// TIA Portal V20 export
FUNCTION_BLOCK "Simulation"   // FB191, LAD
// stored: MemoryReserve 100, Namespace Unit1.Em3, SetENOAutomatically false
   VAR_INPUT
      simulation { ExternalAccessible := 'False'; ExternalVisible := 'False'; ExternalWritable := 'False'} : Bool;
   END_VAR
   VAR
      instActuator { ExternalAccessible := 'False'; ExternalVisible := 'False'; ExternalWritable := 'False'} : Array[0..19] of "Simulation_Actuator";
      statDigitalSignal { ExternalAccessible := 'False'; ExternalVisible := 'False'; ExternalWritable := 'False'} : Array[0..9] of Bool;
   END_VAR
   VAR_TEMP
      tempJRPnPRightplace : Bool;
   END_VAR
   VAR_TEMP   // added for the SCL form of the ladder/FBD networks
      _w1 : Bool;
   END_VAR
BEGIN

REGION Network 1: Digital Signal
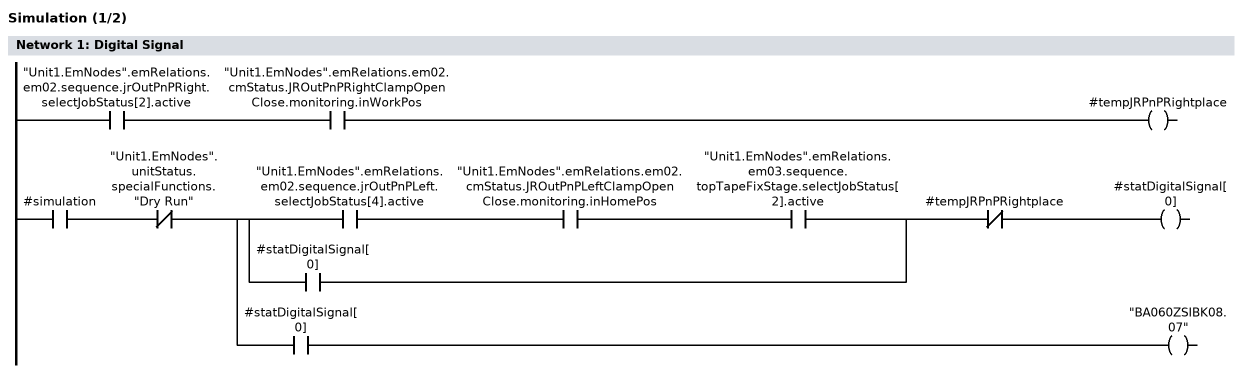
   RUNG wire#powerrail
      Contact( "Unit1.EmNodes".emRelations.em02.sequence.jrOutPnPRight.selectJobStatus[2].active )
      Contact( "Unit1.EmNodes".emRelations.em02.cmStatus.JROutPnPRightClampOpenClose.monitoring.inWorkPos )
      Coil( #tempJRPnPRightplace )
   END_RUNG
   RUNG wire#powerrail
      Contact( #simulation )
      I_Contact( "Unit1.EmNodes".unitStatus.specialFunctions."Dry Run" )
      wire#w1
      Contact( "Unit1.EmNodes".emRelations.em02.sequence.jrOutPnPLeft.selectJobStatus[4].active )
      Contact( "Unit1.EmNodes".emRelations.em02.cmStatus.JROutPnPLeftClampOpenClose.monitoring.inHomePos )
      Contact( "Unit1.EmNodes".emRelations.em03.sequence.topTapeFixStage.selectJobStatus[2].active )
      wire#w2
      I_Contact( #tempJRPnPRightplace )
      Coil( #statDigitalSignal[0] )
   END_RUNG
   RUNG wire#w1
      Contact( #statDigitalSignal[0] )
   END_RUNG wire#w2
   RUNG wire#w1
      Contact( #statDigitalSignal[0] )
      Coil( "BA060ZSIBK08.07" )
   END_RUNG
   // the same network as SCL:
   #tempJRPnPRightplace := "Unit1.EmNodes".emRelations.em02.sequence.jrOutPnPRight.selectJobStatus[2].active AND "Unit1.EmNodes".emRelations.em02.cmStatus.JROutPnPRightClampOpenClose.monitoring.inWorkPos;
   #_w1 := #simulation AND NOT "Unit1.EmNodes".unitStatus.specialFunctions."Dry Run";
   #statDigitalSignal[0] := #_w1 AND (("Unit1.EmNodes".emRelations.em02.sequence.jrOutPnPLeft.selectJobStatus[4].active AND "Unit1.EmNodes".emRelations.em02.cmStatus.JROutPnPLeftClampOpenClose.monitoring.inHomePos AND "Unit1.EmNodes".emRelations.em03.sequence.topTapeFixStage.selectJobStatus[2].active) OR #statDigitalSignal[0]) AND NOT #tempJRPnPRightplace;
   "BA060ZSIBK08.07" := #_w1 AND #statDigitalSignal[0];
END_REGION

REGION Network 2: Two Way Actuator
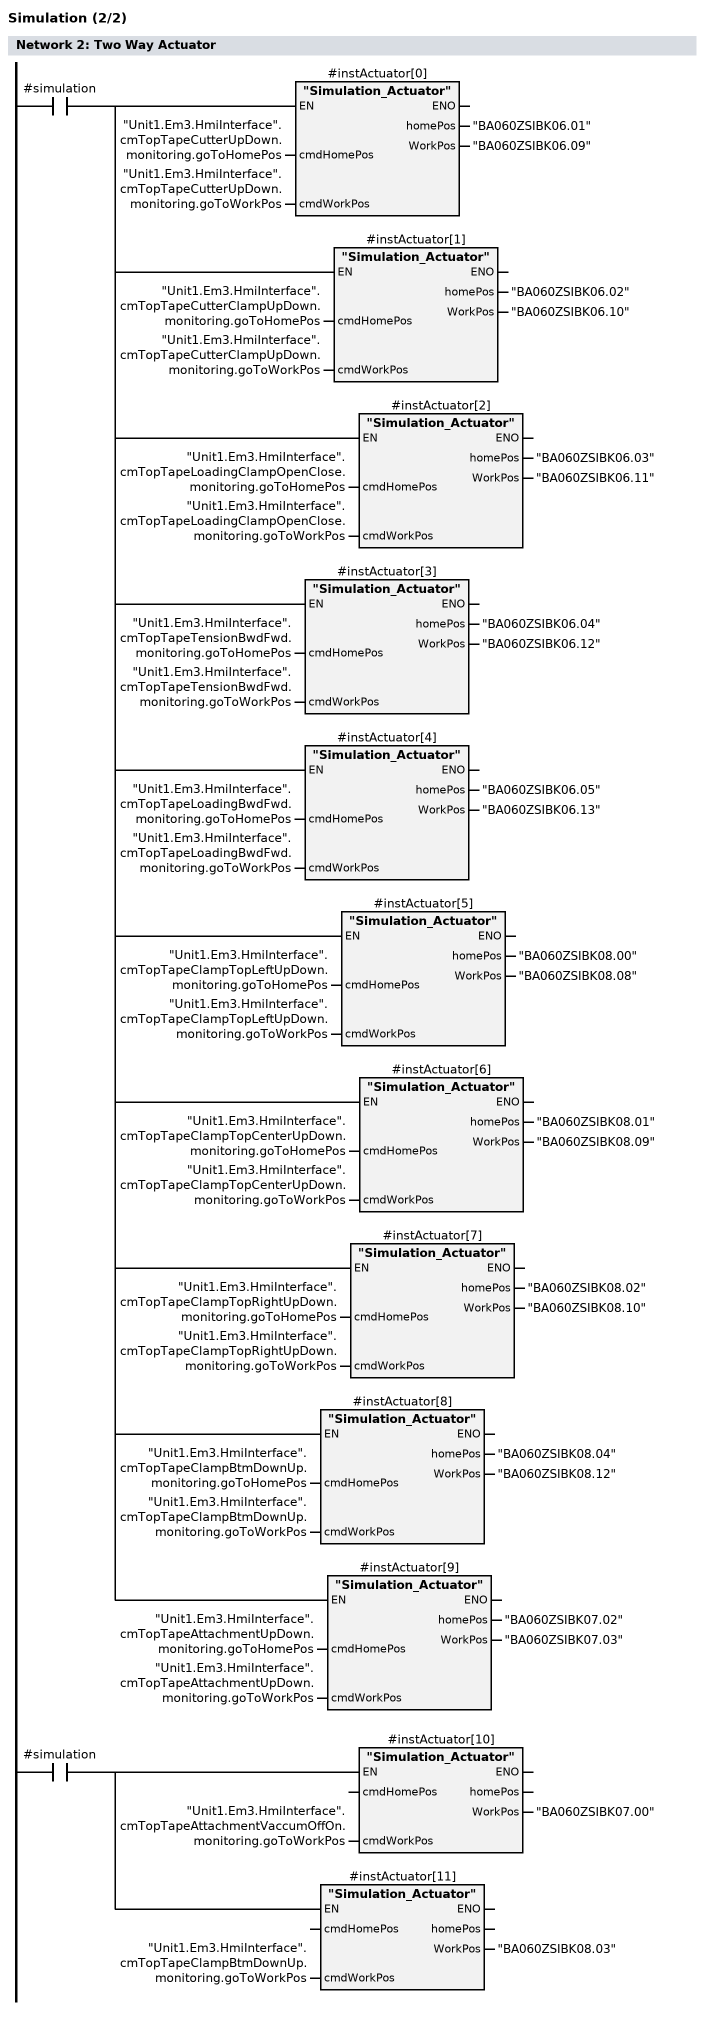
   RUNG wire#powerrail
      Contact( #simulation )
      wire#w1
      #instActuator[0](cmdHomePos := "Unit1.Em3.HmiInterface".cmTopTapeCutterUpDown.monitoring.goToHomePos, cmdWorkPos := "Unit1.Em3.HmiInterface".cmTopTapeCutterUpDown.monitoring.goToWorkPos, homePos => "BA060ZSIBK06.01", WorkPos => "BA060ZSIBK06.09")
   END_RUNG
   RUNG wire#w1
      #instActuator[1](cmdHomePos := "Unit1.Em3.HmiInterface".cmTopTapeCutterClampUpDown.monitoring.goToHomePos, cmdWorkPos := "Unit1.Em3.HmiInterface".cmTopTapeCutterClampUpDown.monitoring.goToWorkPos, homePos => "BA060ZSIBK06.02", WorkPos => "BA060ZSIBK06.10")
   END_RUNG
   RUNG wire#w1
      #instActuator[2](cmdHomePos := "Unit1.Em3.HmiInterface".cmTopTapeLoadingClampOpenClose.monitoring.goToHomePos, cmdWorkPos := "Unit1.Em3.HmiInterface".cmTopTapeLoadingClampOpenClose.monitoring.goToWorkPos, homePos => "BA060ZSIBK06.03", WorkPos => "BA060ZSIBK06.11")
   END_RUNG
   RUNG wire#w1
      #instActuator[3](cmdHomePos := "Unit1.Em3.HmiInterface".cmTopTapeTensionBwdFwd.monitoring.goToHomePos, cmdWorkPos := "Unit1.Em3.HmiInterface".cmTopTapeTensionBwdFwd.monitoring.goToWorkPos, homePos => "BA060ZSIBK06.04", WorkPos => "BA060ZSIBK06.12")
   END_RUNG
   RUNG wire#w1
      #instActuator[4](cmdHomePos := "Unit1.Em3.HmiInterface".cmTopTapeLoadingBwdFwd.monitoring.goToHomePos, cmdWorkPos := "Unit1.Em3.HmiInterface".cmTopTapeLoadingBwdFwd.monitoring.goToWorkPos, homePos => "BA060ZSIBK06.05", WorkPos => "BA060ZSIBK06.13")
   END_RUNG
   RUNG wire#w1
      #instActuator[5](cmdHomePos := "Unit1.Em3.HmiInterface".cmTopTapeClampTopLeftUpDown.monitoring.goToHomePos, cmdWorkPos := "Unit1.Em3.HmiInterface".cmTopTapeClampTopLeftUpDown.monitoring.goToWorkPos, homePos => "BA060ZSIBK08.00", WorkPos => "BA060ZSIBK08.08")
   END_RUNG
   RUNG wire#w1
      #instActuator[6](cmdHomePos := "Unit1.Em3.HmiInterface".cmTopTapeClampTopCenterUpDown.monitoring.goToHomePos, cmdWorkPos := "Unit1.Em3.HmiInterface".cmTopTapeClampTopCenterUpDown.monitoring.goToWorkPos, homePos => "BA060ZSIBK08.01", WorkPos => "BA060ZSIBK08.09")
   END_RUNG
   RUNG wire#w1
      #instActuator[7](cmdHomePos := "Unit1.Em3.HmiInterface".cmTopTapeClampTopRightUpDown.monitoring.goToHomePos, cmdWorkPos := "Unit1.Em3.HmiInterface".cmTopTapeClampTopRightUpDown.monitoring.goToWorkPos, homePos => "BA060ZSIBK08.02", WorkPos => "BA060ZSIBK08.10")
   END_RUNG
   RUNG wire#w1
      #instActuator[8](cmdHomePos := "Unit1.Em3.HmiInterface".cmTopTapeClampBtmDownUp.monitoring.goToHomePos, cmdWorkPos := "Unit1.Em3.HmiInterface".cmTopTapeClampBtmDownUp.monitoring.goToWorkPos, homePos => "BA060ZSIBK08.04", WorkPos => "BA060ZSIBK08.12")
   END_RUNG
   RUNG wire#w1
      #instActuator[9](cmdHomePos := "Unit1.Em3.HmiInterface".cmTopTapeAttachmentUpDown.monitoring.goToHomePos, cmdWorkPos := "Unit1.Em3.HmiInterface".cmTopTapeAttachmentUpDown.monitoring.goToWorkPos, homePos => "BA060ZSIBK07.02", WorkPos => "BA060ZSIBK07.03")
   END_RUNG
   RUNG wire#powerrail
      Contact( #simulation )
      wire#w2
      #instActuator[10](cmdHomePos :=, cmdWorkPos := "Unit1.Em3.HmiInterface".cmTopTapeAttachmentVaccumOffOn.monitoring.goToWorkPos, homePos =>, WorkPos => "BA060ZSIBK07.00")
   END_RUNG
   RUNG wire#w2
      #instActuator[11](cmdHomePos :=, cmdWorkPos := "Unit1.Em3.HmiInterface".cmTopTapeClampBtmDownUp.monitoring.goToWorkPos, homePos =>, WorkPos => "BA060ZSIBK08.03")
   END_RUNG
   // the same network as SCL:
   IF #simulation THEN
       #instActuator[0](cmdHomePos := "Unit1.Em3.HmiInterface".cmTopTapeCutterUpDown.monitoring.goToHomePos,   // "Simulation_Actuator"
                        cmdWorkPos := "Unit1.Em3.HmiInterface".cmTopTapeCutterUpDown.monitoring.goToWorkPos,
                        homePos => "BA060ZSIBK06.01",
                        WorkPos => "BA060ZSIBK06.09");
       #instActuator[1](cmdHomePos := "Unit1.Em3.HmiInterface".cmTopTapeCutterClampUpDown.monitoring.goToHomePos,   // "Simulation_Actuator"
                        cmdWorkPos := "Unit1.Em3.HmiInterface".cmTopTapeCutterClampUpDown.monitoring.goToWorkPos,
                        homePos => "BA060ZSIBK06.02",
                        WorkPos => "BA060ZSIBK06.10");
       #instActuator[2](cmdHomePos := "Unit1.Em3.HmiInterface".cmTopTapeLoadingClampOpenClose.monitoring.goToHomePos,   // "Simulation_Actuator"
                        cmdWorkPos := "Unit1.Em3.HmiInterface".cmTopTapeLoadingClampOpenClose.monitoring.goToWorkPos,
                        homePos => "BA060ZSIBK06.03",
                        WorkPos => "BA060ZSIBK06.11");
       #instActuator[3](cmdHomePos := "Unit1.Em3.HmiInterface".cmTopTapeTensionBwdFwd.monitoring.goToHomePos,   // "Simulation_Actuator"
                        cmdWorkPos := "Unit1.Em3.HmiInterface".cmTopTapeTensionBwdFwd.monitoring.goToWorkPos,
                        homePos => "BA060ZSIBK06.04",
                        WorkPos => "BA060ZSIBK06.12");
       #instActuator[4](cmdHomePos := "Unit1.Em3.HmiInterface".cmTopTapeLoadingBwdFwd.monitoring.goToHomePos,   // "Simulation_Actuator"
                        cmdWorkPos := "Unit1.Em3.HmiInterface".cmTopTapeLoadingBwdFwd.monitoring.goToWorkPos,
                        homePos => "BA060ZSIBK06.05",
                        WorkPos => "BA060ZSIBK06.13");
       #instActuator[5](cmdHomePos := "Unit1.Em3.HmiInterface".cmTopTapeClampTopLeftUpDown.monitoring.goToHomePos,   // "Simulation_Actuator"
                        cmdWorkPos := "Unit1.Em3.HmiInterface".cmTopTapeClampTopLeftUpDown.monitoring.goToWorkPos,
                        homePos => "BA060ZSIBK08.00",
                        WorkPos => "BA060ZSIBK08.08");
       #instActuator[6](cmdHomePos := "Unit1.Em3.HmiInterface".cmTopTapeClampTopCenterUpDown.monitoring.goToHomePos,   // "Simulation_Actuator"
                        cmdWorkPos := "Unit1.Em3.HmiInterface".cmTopTapeClampTopCenterUpDown.monitoring.goToWorkPos,
                        homePos => "BA060ZSIBK08.01",
                        WorkPos => "BA060ZSIBK08.09");
       #instActuator[7](cmdHomePos := "Unit1.Em3.HmiInterface".cmTopTapeClampTopRightUpDown.monitoring.goToHomePos,   // "Simulation_Actuator"
                        cmdWorkPos := "Unit1.Em3.HmiInterface".cmTopTapeClampTopRightUpDown.monitoring.goToWorkPos,
                        homePos => "BA060ZSIBK08.02",
                        WorkPos => "BA060ZSIBK08.10");
       #instActuator[8](cmdHomePos := "Unit1.Em3.HmiInterface".cmTopTapeClampBtmDownUp.monitoring.goToHomePos,   // "Simulation_Actuator"
                        cmdWorkPos := "Unit1.Em3.HmiInterface".cmTopTapeClampBtmDownUp.monitoring.goToWorkPos,
                        homePos => "BA060ZSIBK08.04",
                        WorkPos => "BA060ZSIBK08.12");
       #instActuator[9](cmdHomePos := "Unit1.Em3.HmiInterface".cmTopTapeAttachmentUpDown.monitoring.goToHomePos,   // "Simulation_Actuator"
                        cmdWorkPos := "Unit1.Em3.HmiInterface".cmTopTapeAttachmentUpDown.monitoring.goToWorkPos,
                        homePos => "BA060ZSIBK07.02",
                        WorkPos => "BA060ZSIBK07.03");
       #instActuator[10](cmdWorkPos := "Unit1.Em3.HmiInterface".cmTopTapeAttachmentVaccumOffOn.monitoring.goToWorkPos,   // "Simulation_Actuator"
                         WorkPos => "BA060ZSIBK07.00");
       #instActuator[11](cmdWorkPos := "Unit1.Em3.HmiInterface".cmTopTapeClampBtmDownUp.monitoring.goToWorkPos,   // "Simulation_Actuator"
                         WorkPos => "BA060ZSIBK08.03");
   END_IF;
END_REGION

REGION Network 3 (SCL): homing
   IF #simulation AND "JB_Temp".Test_Homing[3] THEN

       "Unit1.Em3.HmiInterface".cmTopTapeAxisX.commands.homing :=
       "Unit1.Em3.HmiInterface".cmTopTapeAxisY.commands.homing :=
       "Unit1.Em3.HmiInterface".cmTopTapeAttachmentVaccumOffOn.commands.commandHomePos :=
       "Unit1.Em3.HmiInterface".cmTopTapeLoadingBwdFwd.commands.commandWorkPos :=
       "Unit1.Em3.HmiInterface".cmTopTapeLoadingClampOpenClose.commands.commandHomePos :=
       "Unit1.Em3.HmiInterface".cmTopTapeClampAllOpenClose.commands.commandWorkPos := true;
       "Unit1.Em3.HmiInterface".cmTopTapeAttachmentUpDown.commands.commandHomePos := true;


       "JB_Temp".Test_Homing[3] := false;


   END_IF;

   IF #simulation AND "JB_Temp".Test_Homing[20] THEN


       "Unit1.Em3.HmiInterface".cmTopTapeClampAllOpenClose.commands.commandWorkPos :=
       "Unit1.Em3.HmiInterface".cmTopTapeLoadingClampOpenClose.commands.commandHomePos :=
       "Unit1.Em3.HmiInterface".cmTopTapeAxisX.commands.homing :=
       "Unit1.Em3.HmiInterface".cmTopTapeAxisY.commands.homing :=
       "Unit1.Em3.HmiInterface".cmTopTapeAttachmentUpDown.commands.commandHomePos := false;
       "Unit1.Em3.HmiInterface".cmTopTapeLoadingBwdFwd.commands.commandWorkPos := false;

   END_IF;
END_REGION
END_FUNCTION_BLOCK
